PROGRAM PRG_LARS_01_TransportConvCtrl
VAR
	fbPerformance				: FB_Interval;
	tofTransferConvDelay		: FB_TOFR;

END_VAR

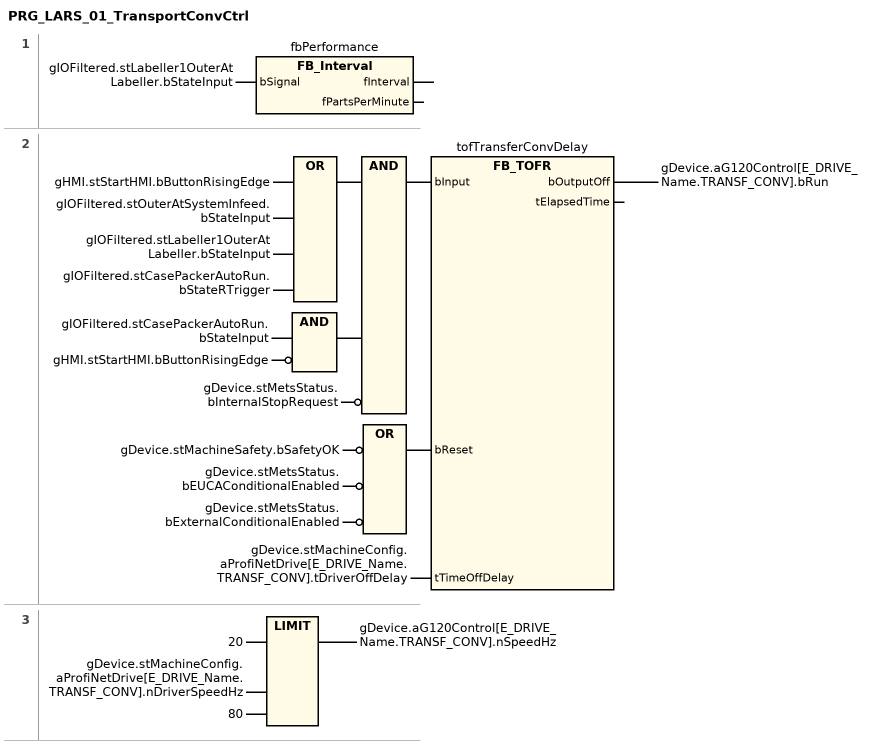
// NETWORK 1
fbPerformance(bSignal := gIOFiltered.stLabeller1OuterAtLabeller.bStateInput); // FB_Interval

// NETWORK 2
tofTransferConvDelay(
    bInput := (gHMI.stStartHMI.bButtonRisingEdge OR gIOFiltered.stOuterAtSystemInfeed.bStateInput OR gIOFiltered.stLabeller1OuterAtLabeller.bStateInput OR gIOFiltered.stCasePackerAutoRun.bStateRTrigger) AND (gIOFiltered.stCasePackerAutoRun.bStateInput AND NOT gHMI.stStartHMI.bButtonRisingEdge) AND NOT gDevice.stMetsStatus.bInternalStopRequest,
    bReset := NOT gDevice.stMachineSafety.bSafetyOK OR NOT gDevice.stMetsStatus.bEUCAConditionalEnabled OR NOT gDevice.stMetsStatus.bExternalConditionalEnabled,
    tTimeOffDelay := gDevice.stMachineConfig.aProfiNetDrive[E_DRIVE_Name.TRANSF_CONV].tDriverOffDelay); // FB_TOFR
gDevice.aG120Control[E_DRIVE_Name.TRANSF_CONV].bRun := tofTransferConvDelay.bOutputOff;

// NETWORK 3
gDevice.aG120Control[E_DRIVE_Name.TRANSF_CONV].nSpeedHz := LIMIT(20, gDevice.stMachineConfig.aProfiNetDrive[E_DRIVE_Name.TRANSF_CONV].nDriverSpeedHz, 80);

END_PROGRAM

(* stored: Version 1.1.0.1
   POU PRG_LARS_01_TransportConvCtrl: Id {9fd5863e-54e1-47d9-9677-b93caeef3e74}, SpecialFunc None *)
